// TIA Portal V20 export
ORGANIZATION_BLOCK "Main"   // OB1, LAD, ProgramCycle
TITLE = "Main Program Sweep (Cycle)"
{ S7_Optimized_Access := 'TRUE' }
// stored: SetENOAutomatically false
   VAR_INPUT
      Initial_Call : Bool;   // Initial call of this OB
      Remanence : Bool;   // =True, if remanent data are available
   END_VAR
BEGIN

REGION Network 1
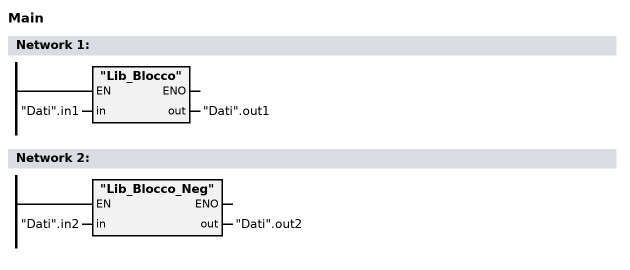
   RUNG wire#powerrail
      "Lib_Blocco"(in := "Dati".in1, out => "Dati".out1)
   END_RUNG
   // the same network as SCL:
   "Lib_Blocco"(in := "Dati".in1, out => "Dati".out1);
END_REGION

REGION Network 2
   RUNG wire#powerrail
      "Lib_Blocco_Neg"(in := "Dati".in2, out => "Dati".out2)
   END_RUNG
   // the same network as SCL:
   "Lib_Blocco_Neg"(in := "Dati".in2, out => "Dati".out2);
END_REGION
END_ORGANIZATION_BLOCK
